% RSLogix 500 project PRACTISE-19.RSS, saved by version 8.30.00.16 %
PROJECT "UNTITLED"    % processor: MicroLogix 1000 %

PROGRAM FILES
  LAD 2 "MAIN_PROG"  5 rungs
  LAD 3 "USER_FAULT"  1 rungs
  LAD 4 "HSC_INT"  1 rungs
  LAD 5 "STI_INT"  1 rungs
  LAD 6, 7, 8, 9, 10, 11, 12, 13, 14, 15, 16: only END

DATA FILES
  O0 OUTPUT  1 elements
  I1 INPUT  2 elements
  S2 STATUS  33 elements
  B3 BINARY  32 elements
  T4 TIMER  40 elements
  C5 COUNTER  32 elements
  R6 CONTROL  16 elements
  N7 INTEGER  105 elements

LADDER 2 "MAIN_PROG"
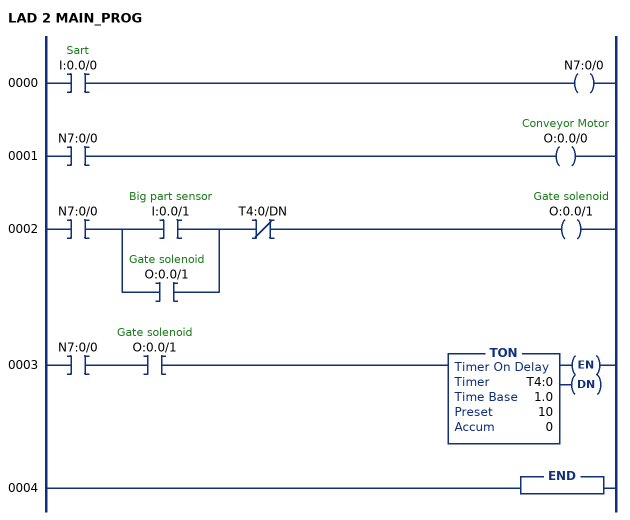
% Rung: 0 %
SOR XIC I:0.0/0 OTE N7:0/0 EOR
%   I:0.0/0  "Sart" %
% Rung: 1 %
SOR XIC N7:0/0 OTE O:0.0/0 EOR
%   O:0.0/0  "Conveyor Motor" %
% Rung: 2 %
SOR XIC N7:0/0 BST XIC I:0.0/1 NXB XIC O:0.0/1 BND XIO T4:0/DN OTE O:0.0/1 EOR
%   I:0.0/1  "Big part sensor" %
%   O:0.0/1  "Gate solenoid" %
% Rung: 3 %
SOR XIC N7:0/0 XIC O:0.0/1 TON T4:0 1.0 10 0 EOR
%   O:0.0/1  "Gate solenoid" %
% Rung: 4 %
SOR END EOR

DATA TABLE (non-zero values as saved)
DATA T4
% .PRE .ACC %
% T4:0 % 10 0
